INTERFACE I_HmiReportable

PROPERTY StatusText : STRING(80)
GET
END_GET
END_PROPERTY

PROPERTY StateNumber : INT
GET
END_GET
END_PROPERTY

PROPERTY AlarmActive : BOOL
GET
END_GET
END_PROPERTY

PROPERTY AlarmMessage : STRING(255)
GET
END_GET
END_PROPERTY

END_INTERFACE

(* stored: Version 1.1.0.1
   Itf I_HmiReportable: Id {3561b024-12f2-4e56-b022-07218a30742a}
   Property StatusText: Id {648f128e-39d0-44fe-8811-633f69f1f762}
   Get Get: Id {ad2f9492-d14a-4e1c-9b95-22f7fe1d21b1}
   Property StateNumber: Id {e2411eb3-9956-4e17-af30-cb2dc2e78aa4}
   Get Get: Id {eaf53e28-24bb-44fd-85d1-1015c8e6619b}
   Property AlarmActive: Id {87093927-0434-4e5e-a374-6a834ab7d185}
   Get Get: Id {0b086a32-434a-445e-9fae-b5401263b2d6}
   Property AlarmMessage: Id {5074ebbb-e87c-4bf9-b7e0-7040a42a9810}
   Get Get: Id {e4a425d6-5a21-4931-994a-6227c8f2f271} *)
